// TIA Portal V18 export
DATA_BLOCK "MAN_DESCRETE_cycle_DB"   // DB32
VERSION : 0.1
// stored: AutoNumber true, DBAccessibleFromOPCUA true, InstanceOfName MAN_DESCRETE_cycle, InstanceOfType FB
"MAN_DESCRETE_cycle"
   // VAR_INPUT
   //    off_conditions : Bool;
   //    on_trigger : Bool;
   // END_VAR
   // VAR_OUTPUT
   //    motors_go_now_command : Bool;
   // END_VAR
   // VAR_IN_OUT
   //    sate : UInt;
   // END_VAR
BEGIN
END_DATA_BLOCK
